{attribute addProperty BoxType "EJ2918-0000-0017"}
{attribute addProperty Id "OutputsOutputs_CA874E89648"}
{attribute addProperty CRC "367035718"}
{attribute addProperty SizeInBites "64"}
{attribute addProperty SizeInBytes "8"}
TYPE Module_2_FSOUT_15E08546 :
STRUCT
	{attribute addProperty Name "Outputs"}
	Outputs  : Outputs_CA874E89;
END_STRUCT
END_TYPE

(* stored: Version 1.2.0.0, ProductVersion 3.1.4024.9
   DUT Module_2_FSOUT_15E08546: Id {9e614b44-07f5-4736-9fc4-a115da1d2977} *)
